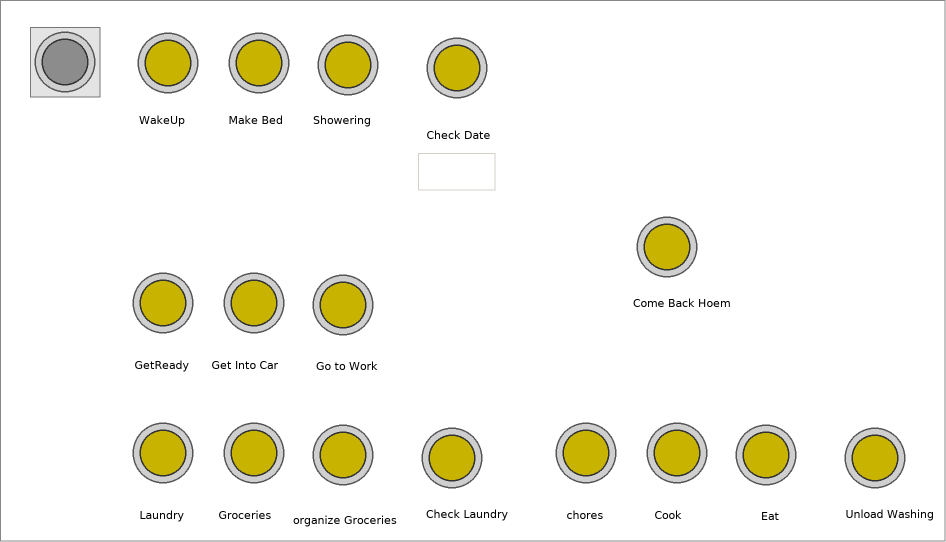
VISUALIZATION Visualization  // 946x542
    Textfield (418,153 77x37), text variable: MAIN.Day
        OnMouseLeave: write the text variable via Edit
    Lamp1 (133,28 70x70), variable: gvl.WakeUp, style: Lamp-Lamp1-Yellow
    Lamp1 (224,28 70x70), variable: gvl.MakeTheBed, style: Lamp-Lamp1-Yellow
    Lamp1 (313,30 70x70), variable: gvl.TakeShower, style: Lamp-Lamp1-Yellow
    Lamp1 (422,33 70x70), variable: gvl.DateCheck, style: Lamp-Lamp1-Yellow
    PushSwitch (30,27 70x70), variable: gvl.Morning, behaviour: TAP, style: Switch-PushSwitch-Gray
    Label (128,103 68x35), "WakeUp"
    Label (420,117 77x37), "Check Date"
    Label (221,103 70x35), "Make Bed"
    Label (308,103 68x35), "Showering"
    Lamp1 (632,212 70x70), variable: GVL.ComeBackHome, style: Lamp-Lamp1-Yellow
    Lamp1 (128,268 70x70), variable: Routine1.GetReadyR1, style: Lamp-Lamp1-Yellow
    Lamp1 (219,268 70x70), variable: Routine1.GetIntoCarR1, style: Lamp-Lamp1-Yellow
    Lamp1 (308,270 70x70), variable: Routine1.GoToworkR1, style: Lamp-Lamp1-Yellow
    Label (128,348 68x35), "GetReady"
    Label (626,286 112x35), "Come Back Hoem"
    Label (313,349 68x35), "Go to Work"
    Label (211,348 68x35), "Get Into Car"
    Lamp1 (417,423 70x70), variable: Routine2.CheckWashingMachineR2, style: Lamp-Lamp1-Yellow
    Lamp1 (128,418 70x70), variable: Routine2.DoLaundriesR2, style: Lamp-Lamp1-Yellow
    Lamp1 (219,418 70x70), variable: Routine2.DoGroceriesR2, style: Lamp-Lamp1-Yellow
    Lamp1 (308,420 70x70), variable: Routine2.OrganizeGroceriesR2, style: Lamp-Lamp1-Yellow
    Label (128,498 68x35), "Laundry"
    Label (411,497 112x35), "Check Laundry"
    Label (282,499 126x43), "organize Groceries"
    Label (211,498 68x35), "Groceries"
    Lamp1 (840,423 70x70), variable: Routine2.UnloadMachineR2, style: Lamp-Lamp1-Yellow
    Lamp1 (551,418 70x70), variable: Routine2.DoOtherChoresR2, style: Lamp-Lamp1-Yellow
    Lamp1 (642,418 70x70), variable: Routine2.CookSomethingR2, style: Lamp-Lamp1-Yellow
    Lamp1 (731,420 70x70), variable: Routine2.EatLunchR2, style: Lamp-Lamp1-Yellow
    Label (551,498 68x35), "chores"
    Label (834,497 112x35), "Unload Washing"
    Label (736,499 68x35), "Eat"
    Label (634,498 68x35), "Cook"
END_VISUALIZATION

(* stored: Version 1.1.0.1, ProductVersion 3.1.4024.12
   Visu Visualization: Id {4ad406ef-aac6-4dea-a62b-4c97dd3af3d8} *)
